(* IEC 61131-3 sources: Std_PalletMover/Class/HandleSteering, 1 file *)

(* ---- HandleSteering.st ---- *)
(*!
<Class
	Name               = "HandleSteering"
	Revision           = "0.0"
	RealtimeTask       = "false"
	CyclicTask         = "false"
	BackgroundTask     = "false"
	Sigmatek           = "false"
	OSInterface        = "false"
	HighPriority       = "false"
	Automatic          = "false"
	UpdateMode         = "Prescan"
	SharedCommandTable = "true"
	Objectsize         = "(562,120)">
	<Channels>
		<Server Name="Actual" Visualized="false" Initialize="false" WriteProtected="true" Retentive="false"/>
		<Server Name="BusyReferencing" Visualized="false" Initialize="false" WriteProtected="true" Retentive="false"/>
		<Server Name="ClassSvr" Visualized="false" Initialize="false" WriteProtected="true" Retentive="false"/>
		<Server Name="IsReferenced" Visualized="false" Initialize="false" WriteProtected="true" Retentive="false"/>
		<Server Name="Setpoint" Visualized="false" Initialize="false" WriteProtected="false" Retentive="false"/>
	</Channels>
</Class>
*)
HandleSteering : CLASS
	TYPE
	  eDriveMode :  //! <Type Public="true" Name="eDriveMode"/>
	  (
	    dm_Idle,
	    dm_Manual,
	    dm_Auto,
	    dm_Referencing,
	    dm_EmergencyStop
	  )$UDINT;
#pragma pack(push, 1)
	  tDriveStatus : STRUCT  //! <Type Public="true" Name="tDriveStatus"/>
	    ds_DriveMode : eDriveMode;
	    ds_Referenced : DINT;
	    ds_Setpoint : REAL;
	    ds_Actual : REAL;
	    ds_FaultCode : DINT;
	    ds_CommunicationOK : DINT;
	    ds_EstopOK : DINT;
	  END_STRUCT;
#pragma pack(pop)
	END_TYPE
  //Servers:
	ClassSvr 	: SvrChCmd_DINT;
	Setpoint 	: SvrCh_REAL;
	Actual 	: SvrCh_REAL;
	IsReferenced 	: SvrCh_DINT;
	BusyReferencing 	: SvrCh_DINT;
  //Clients:
  //Variables:
  //Functions:

	FUNCTION VIRTUAL GLOBAL GetReferenced
		VAR_OUTPUT
			returnValue 	: DINT;
		END_VAR;

	FUNCTION VIRTUAL GLOBAL GetDriveStatus
		VAR_OUTPUT
			returnValue 	: tDriveStatus;
		END_VAR;

	FUNCTION VIRTUAL _forwardSetpoint
		VAR_INPUT
			inputSetpoint 	: REAL;
		END_VAR;

	FUNCTION VIRTUAL _getActual
		VAR_OUTPUT
			returnValue 	: REAL;
		END_VAR;

	FUNCTION VIRTUAL GLOBAL StartReferencing;

	FUNCTION VIRTUAL GLOBAL Setpoint::Write
		VAR_INPUT
			input (EAX) 	: REAL;
		END_VAR
		VAR_OUTPUT
			result (EAX) 	: REAL;
		END_VAR;

	FUNCTION VIRTUAL GLOBAL Actual::Read
		VAR_OUTPUT
			output (EAX) 	: REAL;
		END_VAR;
  //Tables:
	FUNCTION @STD
		VAR_OUTPUT
			ret_code	: CONFSTATES;
		END_VAR;
	FUNCTION GLOBAL TAB @CT_;
END_CLASS;

FUNCTION VIRTUAL GLOBAL HandleSteering::GetReferenced
  #pragma warning(disable: 73);
  #pragma warning(disable: 76);
	VAR_OUTPUT
		returnValue 	: DINT;
	END_VAR
  #pragma warning(default: 73);
  #pragma warning(default: 76);
END_FUNCTION

FUNCTION VIRTUAL GLOBAL HandleSteering::Setpoint::Write
	VAR_INPUT
		input (EAX) 	: REAL;
	END_VAR
	VAR_OUTPUT
		result (EAX) 	: REAL;
	END_VAR

	Setpoint := input;
  _forwardSetpoint(Setpoint);
	result := Setpoint;

END_FUNCTION

FUNCTION VIRTUAL GLOBAL HandleSteering::Actual::Read
	VAR_OUTPUT
		output (EAX) 	: REAL;
	END_VAR

  Actual := _getActual();
	output := Actual;

END_FUNCTION

FUNCTION VIRTUAL GLOBAL HandleSteering::GetDriveStatus
  #pragma warning(disable: 73);
  #pragma warning(disable: 76);
	VAR_OUTPUT
		returnValue 	: tDriveStatus;
	END_VAR
  #pragma warning(default: 73);
  #pragma warning(default: 76);
END_FUNCTION

FUNCTION VIRTUAL HandleSteering::_forwardSetpoint
  #pragma warning(disable: 73);
  #pragma warning(disable: 76);
	VAR_INPUT
		inputSetpoint 	: REAL;
	END_VAR
  #pragma warning(default: 73);
  #pragma warning(default: 76);
END_FUNCTION

FUNCTION VIRTUAL HandleSteering::_getActual
	VAR_OUTPUT
		returnValue 	: REAL;
	END_VAR

  returnValue := Actual;

END_FUNCTION

FUNCTION VIRTUAL GLOBAL HandleSteering::StartReferencing

END_FUNCTION
